{attribute 'GeneratedUsingTerminal: EK1122-0000-0018'}
{attribute addProperty BoxType "EK1122-0000-0018"}
{attribute addProperty Id "Beckhoff_EPP5xxxsub_EK1100EK1100_AB5A94672A_0001_EPP5001_0002_0016EPP5001_09076D6E22A_0002_EPP5101_0002_0016EPP5101_1D9AF86332A_0003_EPP5101_0002_0017EPP5101_1D9AF86332A_0004_EPP5101_0011_0016EPP5101_EE4069E438A_0005_EPP5101_0011_0017EPP5101_EE4069E438A_0006_EPP5101_1002_0016EPP5101_1D9AF86332A_0007_EPP5101_1002_0017EPP5101_1D9AF86332A_0008_EPP5151_0002_0016EPP5151_EE4069E438A_0009_EPP5151_0002_0017EPP5151_EE4069E438"}
{attribute addProperty CRC "1804412731"}
{attribute addProperty Size "304"}
TYPE Beckhoff_EPP5xxxEK1122_6B8D273B EXTENDS EK1122_AB5A9467 :
STRUCT
	{attribute addProperty Name "Beckhoff_EPP5xxxsub_EK1100"}
	{attribute addProperty PreviousPort "Beckhoff EPP5xxxEK1122 : D"}
	Beckhoff_EPP5xxxsub_EK1100 : EK1100_AB5A9467;
	{attribute addProperty Name "A_0001_EPP5001_0002_0016"}
	{attribute addProperty PreviousPort "Beckhoff EPP5xxxsub EK1100 : C"}
	A_0001_EPP5001_0002_0016 : EPP5001_09076D6E;
	{attribute addProperty Name "A_0002_EPP5101_0002_0016"}
	{attribute addProperty PreviousPort "A_0001(EPP5001-0002-0016) : B"}
	A_0002_EPP5101_0002_0016 : EPP5101_1D9AF863;
	{attribute addProperty Name "A_0003_EPP5101_0002_0017"}
	{attribute addProperty PreviousPort "A_0002(EPP5101-0002-0016) : B"}
	A_0003_EPP5101_0002_0017 : EPP5101_1D9AF863;
	{attribute addProperty Name "A_0004_EPP5101_0011_0016"}
	{attribute addProperty PreviousPort "A_0003(EPP5101-0002-0017) : B"}
	A_0004_EPP5101_0011_0016 : EPP5101_EE4069E4;
	{attribute addProperty Name "A_0005_EPP5101_0011_0017"}
	{attribute addProperty PreviousPort "A_0004(EPP5101-0011-0016) : B"}
	A_0005_EPP5101_0011_0017 : EPP5101_EE4069E4;
	{attribute addProperty Name "A_0006_EPP5101_1002_0016"}
	{attribute addProperty PreviousPort "A_0005(EPP5101-0011-0017) : B"}
	A_0006_EPP5101_1002_0016 : EPP5101_1D9AF863;
	{attribute addProperty Name "A_0007_EPP5101_1002_0017"}
	{attribute addProperty PreviousPort "A_0006(EPP5101-1002-0016) : B"}
	A_0007_EPP5101_1002_0017 : EPP5101_1D9AF863;
	{attribute addProperty Name "A_0008_EPP5151_0002_0016"}
	{attribute addProperty PreviousPort "A_0007(EPP5101-1002-0017) : B"}
	A_0008_EPP5151_0002_0016 : EPP5151_EE4069E4;
	{attribute addProperty Name "A_0009_EPP5151_0002_0017"}
	{attribute addProperty PreviousPort "A_0008(EPP5151-0002-0016) : B"}
	A_0009_EPP5151_0002_0017 : EPP5151_EE4069E4;
END_STRUCT
END_TYPE

(* stored: Version 1.2.0.0, ProductVersion 3.1.4024.9
   DUT Beckhoff_EPP5xxxEK1122_6B8D273B: Id {86b9b847-78a1-4e13-93a0-6e15e2d65baf} *)
